(****************************************************************
NAME:			FB_PowerOn
DATA:			2017.2.16
VERSION:		1.0.0
DESCRIPTION:	FB_PowerOn
HISTORY:
				2017.2.16		NEW
				2022.10.18 加入Phase两轴

***************************************************************)
FUNCTION_BLOCK FB_Power
VAR_INPUT
	On:BOOL;
	Off:BOOL;
	Check:BOOL;
END_VAR
VAR_OUTPUT
	FbID:DINT:=1001;
	OnState:DINT;
	OffState: INT;
	OnBusy:BOOL;
	OffBusy:BOOL;
	OnStatus:BOOL;
	OffStatus: BOOL;
	Error:BOOL;
	ErrorID:DINT;
	PowerState:DINT;
END_VAR
VAR
	LeftTopLin_MC_Power: MC_Power;
	RightTopLin_MC_Power: MC_Power;
	LeftBottomLin_MC_Power: MC_Power;
	RightBottomLin_MC_Power: MC_Power;
	PhaseUpperLin_MC_Power: MC_Power;
	PhaseLowerLin_MC_Power: MC_Power;
	fb_ton:TON;
END_VAR

(*power on *)
IF On AND NOT Off THEN
	A_PowerOn();
(*Power Off *)
ELSIF Off AND NOT On THEN
	A_PowerOff();
END_IF
(*Check*)
IF Check THEN
	A_CheckPowerStatus();
END_IF

ACTION A_CheckPowerStatus:
A_PowerMC();
IF  LeftTopLin_MC_Power.Status AND RightTopLin_MC_Power.Status
		AND LeftBottomLin_MC_Power.Status AND RightBottomLin_MC_Power.Status
		AND PhaseUpperLin_MC_Power.Status AND PhaseLowerLin_MC_Power.Status THEN
	PowerState:=1;
ELSIF NOT LeftTopLin_MC_Power.Status AND NOT RightTopLin_MC_Power.Status
		AND NOT LeftBottomLin_MC_Power.Status AND NOT RightBottomLin_MC_Power.Status
		AND NOT PhaseUpperLin_MC_Power.Status AND NOT PhaseLowerLin_MC_Power.Status THEN
	PowerState:=0;
ELSE
	PowerState:=-100;
	Error:=TRUE;
	ErrorID:=77;
	(*FB_PlcEmergencyStop();*)
END_IF
END_ACTION

ACTION A_PowerMC:
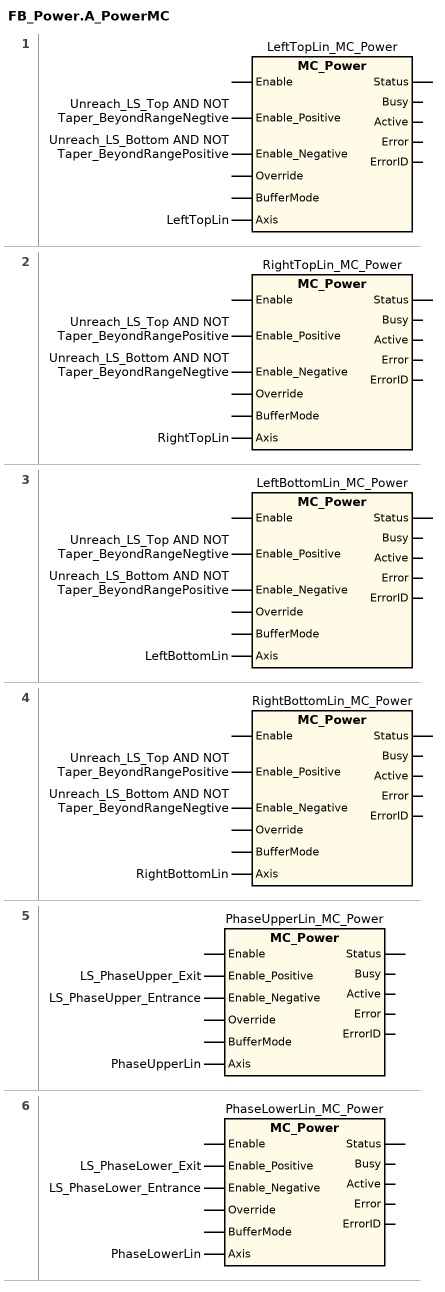
// NETWORK 1
LeftTopLin_MC_Power(
    Enable_Positive := Unreach_LS_Top AND NOT Taper_BeyondRangeNegtive,
    Enable_Negative := Unreach_LS_Bottom AND NOT Taper_BeyondRangePositive,
    Axis := LeftTopLin); // MC_Power

// NETWORK 2
RightTopLin_MC_Power(
    Enable_Positive := Unreach_LS_Top AND NOT Taper_BeyondRangePositive,
    Enable_Negative := Unreach_LS_Bottom AND NOT Taper_BeyondRangeNegtive,
    Axis := RightTopLin); // MC_Power

// NETWORK 3
LeftBottomLin_MC_Power(
    Enable_Positive := Unreach_LS_Top AND NOT Taper_BeyondRangeNegtive,
    Enable_Negative := Unreach_LS_Bottom AND NOT Taper_BeyondRangePositive,
    Axis := LeftBottomLin); // MC_Power

// NETWORK 4
RightBottomLin_MC_Power(
    Enable_Positive := Unreach_LS_Top AND NOT Taper_BeyondRangePositive,
    Enable_Negative := Unreach_LS_Bottom AND NOT Taper_BeyondRangeNegtive,
    Axis := RightBottomLin); // MC_Power

// NETWORK 5
PhaseUpperLin_MC_Power(
    Enable_Positive := LS_PhaseUpper_Exit,
    Enable_Negative := LS_PhaseUpper_Entrance,
    Axis := PhaseUpperLin); // MC_Power

// NETWORK 6
PhaseLowerLin_MC_Power(
    Enable_Positive := LS_PhaseLower_Exit,
    Enable_Negative := LS_PhaseLower_Entrance,
    Axis := PhaseLowerLin); // MC_Power
END_ACTION

ACTION A_PowerOff:
OffBusy:=TRUE;
CASE OffState OF
	0:
		IF NOT LeftTopLin_MC_Power.Status AND NOT RightTopLin_MC_Power.Status
			AND NOT LeftBottomLin_MC_Power.Status AND NOT RightBottomLin_MC_Power.Status 
			AND NOT PhaseUpperLin_MC_Power.Status AND NOT PhaseLowerLin_MC_Power.Status THEN	(*¶¼Ã»ÉÏµç*)
			OffState:=88;
		ELSE
			OffState:=1;
		END_IF
	1:
		LeftTopLin_MC_Power.Enable:=FALSE;
		RightTopLin_MC_Power.Enable:=FALSE;
		LeftBottomLin_MC_Power.Enable:=FALSE;
		RightBottomLin_MC_Power.Enable:=FALSE;
		PhaseUpperLin_MC_Power.Enable:=FALSE;
		PhaseLowerLin_MC_Power.Enable:=FALSE;
		A_PowerMC();
		OffState:=2;
	2:
		IF NOT LeftTopLin_MC_Power.Status AND NOT RightTopLin_MC_Power.Status
			AND NOT LeftBottomLin_MC_Power.Status AND NOT RightBottomLin_MC_Power.Status 
			AND NOT PhaseUpperLin_MC_Power.Status AND NOT PhaseLowerLin_MC_Power.Status THEN	(*¶¼Ã»ÉÏµç*)
			OffState:=88;
		ELSE
			ErrorId:=11;
			OffState:=-100;
		END_IF
	88:
		Off:=FALSE;
		OffState:=0;
		OffBusy:=FALSE;
		OnStatus:=FALSE;
		OffStatus:=TRUE;
		Error:=FALSE;
		ErrorID:=0;
	-100:
		FB_PlcEmergencyStop();
		Off:=FALSE;
		OffState:=-100;
		OffBusy:=FALSE;
		OffStatus:=FALSE;
		Error:=TRUE;

END_CASE
END_ACTION

ACTION A_PowerOn:
OnBusy:=TRUE;
fb_ton(PT:=t#0.5s);
CASE OnState OF
	0:	(*Check*)
		A_PowerMC();
		IF LeftTopLin_MC_Power.Error OR RightTopLin_MC_Power.Error
			OR LeftBottomLin_MC_Power.Error OR RightBottomLin_MC_Power.Error
			OR PhaseUpperLin_MC_Power.Error OR PhaseLowerLin_MC_Power.Error
			OR NOT LeftTopLin_MC_Power.Active OR NOT RightTopLin_MC_Power.Active
			OR NOT LeftBottomLin_MC_Power.Active OR NOT RightBottomLin_MC_Power.Active 
			OR NOT PhaseUpperLin_MC_Power.Active OR NOT PhaseLowerLin_MC_Power.Active THEN		(*FB Error*)
			ErrorID:=1;
			OnState:=99;
		ELSIF LeftTopLin_MC_Power.Status OR RightTopLin_MC_Power.Status
			OR LeftBottomLin_MC_Power.Status OR RightBottomLin_MC_Power.Status 
			OR PhaseUpperLin_MC_Power.Status OR PhaseLowerLin_MC_Power.Status THEN		(*ÖáÒÑ¾­¶¼PowerOn£¬²»·ûºÏ¹¦ÄÜ¿éµ÷ÓÃÌõ¼þ*)
			ErrorID:=2;
			OnState:=-100;
		ELSIF NOT LeftTopLin_MC_Power.Status OR NOT RightTopLin_MC_Power.Status
			OR NOT LeftBottomLin_MC_Power.Status OR NOT RightBottomLin_MC_Power.Status 
			OR NOT PhaseUpperLin_MC_Power.Status OR NOT PhaseLowerLin_MC_Power.Status THEN		(*Öá¶¼Ã»ÓÐPower£¬×ªÏÂÒ»²½*)
			OnState:=1;
		ELSE
			ErrorID:=3;
			OnState:=-100;
		END_IF
	1:	(*Execute*)
		IF NOT LeftTopLin_MC_Power.Status OR NOT RightTopLin_MC_Power.Status
			OR NOT LeftBottomLin_MC_Power.Status OR NOT RightBottomLin_MC_Power.Status 
			OR NOT PhaseUpperLin_MC_Power.Status OR NOT PhaseLowerLin_MC_Power.Status THEN		(*ÔÙ¼ì²é£¬Öá¶¼Ã»ÓÐPower*)
			LeftTopLin_MC_Power.Enable:=TRUE;
			RightTopLin_MC_Power.Enable:=TRUE;
			LeftBottomLin_MC_Power.Enable:=TRUE;
			RightBottomLin_MC_Power.Enable:=TRUE;
			PhaseUpperLin_MC_Power.Enable:=TRUE;
			PhaseLowerLin_MC_Power.Enable:=TRUE;
			A_PowerMC();
			fb_ton.IN:=TRUE;
			OnState:=2;
		ELSE
			ErrorID:=4;
			OnState:=-100;
		END_IF
	2:	(*Wait*)
		A_PowerMC();
		IF NOT LeftTopLin_MC_Power.Status OR NOT RightTopLin_MC_Power.Status
			OR NOT LeftBottomLin_MC_Power.Status OR NOT RightBottomLin_MC_Power.Status 
			OR NOT PhaseUpperLin_MC_Power.Status OR NOT PhaseLowerLin_MC_Power.Status THEN		(*Power StatusÐÅºÅ²»µ½£¬¼ÌÐøµÈ´ý£¬Èç¹û³¬Ê±ÔòFB Error*)
			IF NOT fb_ton.Q THEN
				OnState:=2;
			ELSE
				ErrorID:=8;
				OnState:=99;
			END_IF
		ELSIF  LeftTopLin_MC_Power.Status AND RightTopLin_MC_Power.Status
			AND LeftBottomLin_MC_Power.Status AND RightBottomLin_MC_Power.Status 
			AND PhaseUpperLin_MC_Power.Status AND PhaseLowerLin_MC_Power.Status THEN			(*ÕýÈ·µç»úÉÏµã×´Ì¬£¬×ªÏÂÒ»²½*)
				OnState:=88;
		ELSE
				ErrorID:=9;
				OnState:=-100;
		END_IF
	88:
		On:=FALSE;
		OnState:=0;
		OnBusy:=FALSE;
		OnStatus:=TRUE;
		OffStatus:=FALSE;
		Error:=FALSE;
		ErrorID:=0;
		fb_ton.IN:=FALSE;
	99:
		On:=FALSE;
		OnState:=99;
		OnBusy:=FALSE;
		OnStatus:=FALSE;
		Error:=TRUE;
		LeftTopLin_MC_Power.Enable:=FALSE;
		RightTopLin_MC_Power.Enable:=FALSE;
		LeftBottomLin_MC_Power.Enable:=FALSE;
		RightBottomLin_MC_Power.Enable:=FALSE;
		PhaseUpperLin_MC_Power.Enable:=FALSE;
		PhaseLowerLin_MC_Power.Enable:=FALSE;
		fb_ton.IN:=FALSE;
	-100:
		FB_PlcEmergencyStop();
		On:=FALSE;
		OnState:=-100;
		OnBusy:=FALSE;
		OnStatus:=FALSE;
		Error:=TRUE;
		LeftTopLin_MC_Power.Enable:=FALSE;
		RightTopLin_MC_Power.Enable:=FALSE;
		LeftBottomLin_MC_Power.Enable:=FALSE;
		RightBottomLin_MC_Power.Enable:=FALSE;
		PhaseUpperLin_MC_Power.Enable:=FALSE;
		PhaseLowerLin_MC_Power.Enable:=FALSE;
		fb_ton.IN:=FALSE;

END_CASE
END_ACTION

END_FUNCTION_BLOCK

(* stored: Version 1.1.0.1, ProductVersion 3.1.4024.6
   POU FB_Power: Id {d3a7443c-2919-46ae-a7ad-f8f713ca36af}, SpecialFunc None
   Action A_CheckPowerStatus: Id {45ab49c5-f74b-4ae0-bfbf-f6d250f649c1}
   Action A_PowerMC: Id {d3c8aed1-becd-49d1-b5d2-31e3edecaf6a}
   Action A_PowerOff: Id {f8455d76-f208-4ad8-b331-bf9b4a5057da}
   Action A_PowerOn: Id {46ba4774-a9a2-4a51-9400-f8277a7731df} *)
